// TIA Portal V21 export
ORGANIZATION_BLOCK "MODULE_ERROR_MOLDE"   // OB123, LAD, ProgramCycle
TITLE = MODULE_ERROR_MOLDE
{ S7_Optimized_Access := 'TRUE' }
VERSION : 0.1
// stored: AutoNumber true, IsIECCheckEnabled false, SetENOAutomatically false
   VAR_INPUT
      Initial_Call : Bool;
      Remanence : Bool;
   END_VAR
BEGIN

REGION Network 1: Molde: falha modulo HW 999
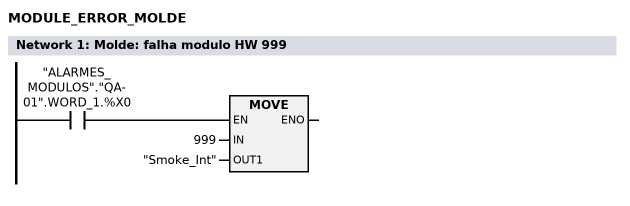
   RUNG wire#powerrail
      Contact( "ALARMES_MODULOS"."QA-01".WORD_1.%X0 )
      { S7_GenerateENO := "TRUE" } Move(in := 999, out1 := "Smoke_Int")
   END_RUNG
   // the same network as SCL:
   IF "ALARMES_MODULOS"."QA-01".WORD_1.%X0 THEN <??.?> := 999; END_IF;
END_REGION
END_ORGANIZATION_BLOCK
